{attribute 'qualified_only'}
{attribute 'strict'}
TYPE E_PNEU_VAC_VALVE :
(
	VacDetect,
	Vac_ON_NotDetect,
	AllOff,
	Blowing
);
END_TYPE

(* stored: Version 1.1.0.1, ProductVersion 3.1.4024.12
   DUT E_PNEU_VAC_VALVE: Id {72614da2-b894-438d-9ce1-811307635741} *)
